(* IEC 61131-3 sources: CodesysTest/export/SX_1195.dev/Plc Logic/Application/PRJ Specific/1195 Testing/Cycle_Rate_Mods/FB_1195_Test_BagDelivery.pou/ReadyForPrint.prop, 1 file *)

(* ---- Get.pm.st ---- *)
(*#-#-#-#-#-#-#-#-#-#---Declaration---#-#-#-#-#-#-#-#-#-#-#-#-#*)

VAR
END_VAR
(*#-#-#-#-#-#-#-#-#-#---Implementation---#-#-#-#-#-#-#-#-#-#-#-#-#*)

ReadyForPrint:= _readyForPrint;
